(* PLC project SafeLOGIC, BrAutomation SafeDESIGNER  5.24.1.0 *)
(* stored: companyURL http://www.br-automation.com, creationDateTime Wed Nov 26 14:27:06 2025 *)

PROGRAM ELAPSED_TIME_TOF

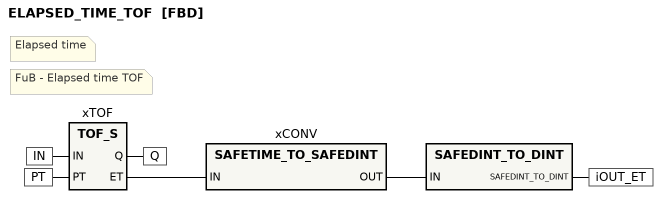
(* FBD diagram, written out as Structured Text *)
(* FuB - Elapsed time TOF *)
(* Elapsed time *)
xTOF(IN := IN, PT := PT);
Q := xTOF.Q;
xCONV(IN := xTOF.ET);
iOUT_ET := SAFEDINT_TO_DINT(xCONV.OUT);
END_PROGRAM
